% RSLogix 500 project TEST3_BAK012.RSS, saved by version 11.00.00.00 %
PROJECT "UNTITLED"    % processor: MicroLogix 1200 %

PROGRAM FILES
  LAD 2 "MAIN_PROG"  13 rungs

DATA FILES
  O0 OUTPUT  4 elements
  I1 INPUT  4 elements
  S2 STATUS  66 elements
  B3 BINARY  1 elements
  T4 TIMER  1 elements
  C5 COUNTER  1 elements
  R6 CONTROL  1 elements
  N7 INTEGER  1 elements
  F8   1 elements

LADDER 2 "MAIN_PROG"
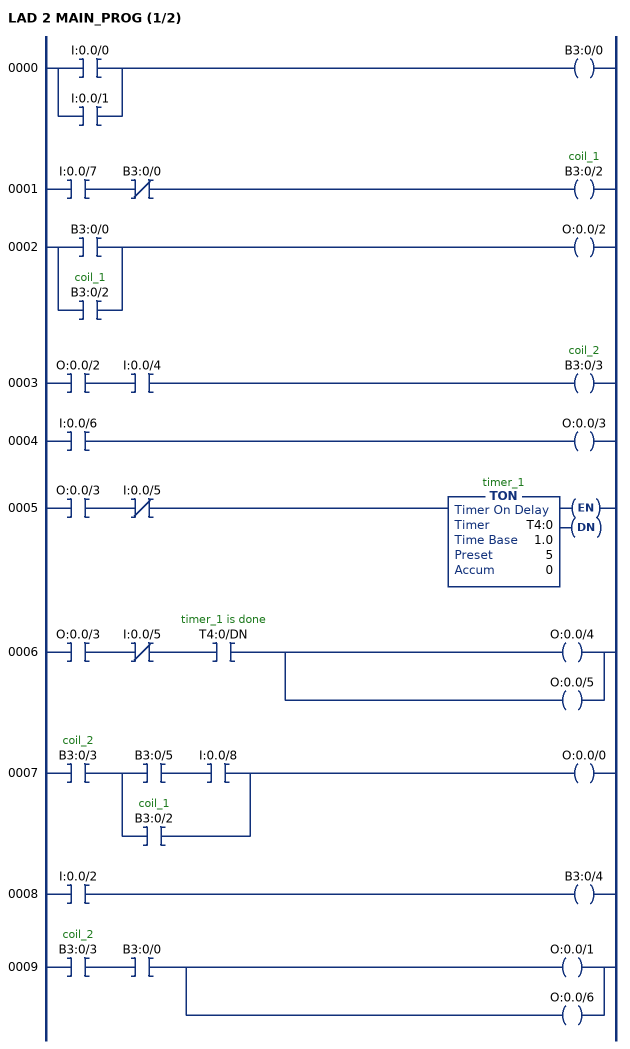
% Rung: 0 %
SOR BST XIC I:0.0/0 NXB XIC I:0.0/1 BND OTE B3:0/0 EOR
% Rung: 1 %
SOR XIC I:0.0/7 XIO B3:0/0 OTE B3:0/2 EOR
%   B3:0/2  "coil_1" %
% Rung: 2 %
SOR BST XIC B3:0/0 NXB XIC B3:0/2 BND OTE O:0.0/2 EOR
%   B3:0/2  "coil_1" %
% Rung: 3 %
SOR XIC O:0.0/2 XIC I:0.0/4 OTE B3:0/3 EOR
%   B3:0/3  "coil_2" %
% Rung: 4 %
SOR XIC I:0.0/6 OTE O:0.0/3 EOR
% Rung: 5 %
SOR XIC O:0.0/3 XIO I:0.0/5 TON T4:0 1.0 5 0 EOR
%   T4:0  "timer_1" %
% Rung: 6 %
SOR XIC O:0.0/3 XIO I:0.0/5 XIC T4:0/DN BST OTE O:0.0/4 NXB OTE O:0.0/5 BND EOR
%   T4:0/DN  "timer_1 is done" %
% Rung: 7 %
SOR XIC B3:0/3 BST XIC B3:0/5 XIC I:0.0/8 NXB XIC B3:0/2 BND OTE O:0.0/0 EOR
%   B3:0/3  "coil_2" %
%   B3:0/2  "coil_1" %
% Rung: 8 %
SOR XIC I:0.0/2 OTE B3:0/4 EOR
% Rung: 9 %
SOR XIC B3:0/3 XIC B3:0/0 BST OTE O:0.0/1 NXB OTE O:0.0/6 BND EOR
%   B3:0/3  "coil_2" %

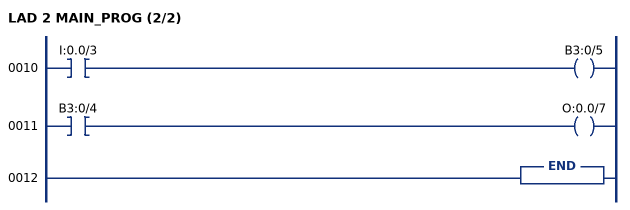
% Rung: 10 %
SOR XIC I:0.0/3 OTE B3:0/5 EOR
% Rung: 11 %
SOR XIC B3:0/4 OTE O:0.0/7 EOR
% Rung: 12 %
SOR END EOR

OTHER DOCUMENTED ADDRESSES
  B3:0  "pb_1"
  B3:0/1  "pb_2"

DATA TABLE (non-zero values as saved)
DATA T4
% .PRE .ACC %
% T4:0 % 5 0
